Staubli VAL3: modIMM.dtx

num nCaseBtRobOff
num nStateRstPart[4]
num nStatePartMade
num reactionTime
num pointer
num timings[40]
public num nCloseDelayTime
num mouldTimer
bool bRobotOffAllow
bool bState
num tmMotionStack
num WAR_MOTIONSTACK = 1
bool bDisplayed
bool bSuspendForTest
num WAIT_MOULD_FREE
num nAreaTestState
num nMouldAreaZone
num WAIT_MOULD_OPEN
num WAIT_ROB_ENABLE
num WAIT_IMM_AUTO
num WAIT_PARTMADE
public string name = "IMM"
num moduleIndex
bool bAtWaitPosition
string IMM_IO_PTH
num nImmType
bool bRobotOff
num AREA_TEST_FAIL
num nMouldAreaDist
num HOME_IN_MOULD
num ARM_IN_MOULD_NO
num ARM_IN_MOULD_ST
